{attribute 'GeneratedUsingTerminal: EL5101-0010-0016'}
{attribute addProperty BoxType "EL5101-0010-0016"}
{attribute addProperty Id "ENC_Status_compactAT %I*ENC_Status_compact_4198EF3B17ENC_Control_compactAT %Q*ENC_Control_compact_21E2D14D6WcStateAT %I*WcState_9091E0EB2InfoDataAT %I*InfoData_94A18F5E2"}
{attribute addProperty CRC "2702897132"}
{attribute addProperty Size "27"}
TYPE EL5101_A11AEFEC EXTENDS EtcSlaveTerminalBase_947E5A46 :
STRUCT
	{attribute addProperty Name "ENC_Status_compact"}
	ENC_Status_compact : ENC_Status_compact_4198EF3B;
	{attribute addProperty Name "ENC_Control_compact"}
	ENC_Control_compact : ENC_Control_compact_21E2D14D;
	{attribute addProperty Name "WcState"}
	WcState : WcState_9091E0EB;
	{attribute addProperty Name "InfoData"}
	InfoData : InfoData_94A18F5E;
END_STRUCT
END_TYPE

(* stored: Version 1.2.0.0, ProductVersion 3.1.4024.9
   DUT EL5101_A11AEFEC: Id {bd668845-ce36-489b-bd92-4445d1a9b671} *)
